TYPE ST_Syntax_Derived EXTENDS ST_Syntax_Mini :
    STRUCT
        fExtendedValue : LREAL      := 3.14159;
        sDescription   : STRING(80) := 'Derived Struct';
        bDerivedActive : BOOL;
    END_STRUCT
END_TYPE

(* stored: Version 1.1.0.1, ProductVersion 3.1.4024.16
   DUT ST_Syntax_Derived: Id {a5da701b-1a78-4251-91bd-8bb3f15fddee} *)
